FUNCTION RFID_Sensor_Read : RFID_Sensor_Error
VAR_INPUT
END_VAR
VAR
END_VAR

END_FUNCTION

(* stored: Version 1.1.0.1, ProductVersion 3.1.4024.10
   POU RFID_Sensor_Read: Id {c3ae08fd-2472-4db9-a318-2e9d26a190f8}, SpecialFunc None *)
